// TIA Portal project "lab3" (V15)

(* hardware
DEVICE "S71500/ET200MP station_1"  S7-1500 station
   slot 0: "Rail_0"  Rack  6ES7 590-1***0-0AA0
   slot 1: "PLC_1"  CPU 1512C-1 PN  6ES7 512-1CK01-0AB0  V2.5
      slot 3: "CPU display_1"  6ES7591-1AA00-0AA0
*)

// ===== PLC "PLC_1"  CPU 1512C-1 PN =====

VAR_GLOBAL   // PLC tag table "Default tag table"
   "DIGITALNI_ULAZ_KLIP_1_LEVO_NC" AT %I10.0 : Bool;
   "DIGITALNI_ULAZ_KLIP_1_DESNO_NC" AT %I10.1 : Bool;
   "DIGITALNI_ULAZ_KLIP_2_LEVO_NO" AT %I10.2 : Bool;
   "DIGITALNI_ULAZ_KLIP_2_DESNO_NC" AT %I10.3 : Bool;
   "DIGITALNI_ULAZ_KLIP_3_LEVO_NO" AT %I10.4 : Bool;
   "DIGITALNI_ULAZ_KLIP_3_DESNO_NO" AT %I10.5 : Bool;
   "DIGITALNI_ULAZ_KLIP_4_LEVO_NC" AT %I10.6 : Bool;
   "DIGITALNI_ULAZ_KLIP_4_DESNO_NO" AT %I10.7 : Bool;
   "DIGITALNI_IZLAZ_KLIP_1_LEVO" AT %Q4.0 : Bool;
   "DIGITALNI_IZLAZ_KLIP_1_DESNO" AT %Q4.1 : Bool;
   "DIGITALNI_IZLAZ_KLIP_2_LEVO" AT %Q4.2 : Bool;
   "DIGITALNI_IZLAZ_KLIP_2_DESNO" AT %Q4.3 : Bool;
   "DIGITALNI_IZLAZ_KLIP_3_LEVO" AT %Q4.4 : Bool;
   "DIGITALNI_IZLAZ_KLIP_4_LEVO" AT %Q4.6 : Bool;
   "ANALOGNI_ULAZ_POZICIJA_KLIP_1" AT %IW0 : Word;
   "ANALOGNI_ULAZ_POZICIJA_KLIP_4" AT %IW2 : Word;
   "TIMER" AT %T0 : Timer;
   "COUNTER_INNER_LOOP" AT %C0 : Counter;
   "COUNTER_OUTER_LOOP" AT %C1 : Counter;
   "BROJAC_ODRZAVANJE_KLIP_4" AT %C2 : Counter;
END_VAR

DATA_BLOCK "DB"   // DB1
{ S7_Optimized_Access := 'TRUE' }
VERSION : 0.1
   VAR
      "POZICIJA_KLIP_30%" : Word := 8310;
      "POZICIJA_KLIP_40%" : Word := 11080;
      "POZICIJA_KLIP_50%" : Word := 13850;
      "POZICIJA_KLIP_70%" : Word := 19390;
      "POZICIJA_KLIP_90%" : Word := 24930;
      "POZICIJA_KLIP_80%" : Word := 22160;
      POZICIJA_MAX : Word := 27700;
   END_VAR
BEGIN
END_DATA_BLOCK

DATA_BLOCK "SEKVENCA_DB"   // DB2
{ S7_Optimized_Access := 'TRUE' }
VERSION : 0.1
// stored: InstanceOfName SEKVENCA
"SEKVENCA"
BEGIN
END_DATA_BLOCK

FUNCTION_BLOCK "SEKVENCA"   // FB1, GRAPH_PLUS
{ S7_Optimized_Access := 'TRUE' }
VERSION : 0.1
   VAR_INPUT
      OFF_SQ : Bool := false;   // Turn sequence off
      INIT_SQ : Bool := false;   // Set sequence to initial state
      ACK_EF : Bool := false;   // Acknowledge all errors and faults
      S_PREV : Bool := false;   // Output previous step in parameter S_NO
      S_NEXT : Bool := false;   // Indicate next step in parameter S_NO
      SW_AUTO : Bool := false;   // Automatic mode
      SW_TAP : Bool := false;   // Semiautomatic/switch with transition
      SW_TOP : Bool := false;   // Semiautomatic/ignore transition
      SW_MAN : Bool := false;   // Manual mode
      S_SEL : Int := 0;   // Select step to be output to S_NO
      S_ON : Bool := false;   // Activate step indicated in S_NO
      S_OFF : Bool := false;   // Deactivate step indicated S_NO
      T_PUSH : Bool := false;   // Enable transition to switch in semi automatic mode
   END_VAR
   VAR_OUTPUT
      S_NO : Int := 0;   // Step number
      S_MORE : Bool := false;   // More steps are available and can be shown in S_NO
      S_ACTIVE : Bool := false;   // Step indicated in S_NO is active
      ERR_FLT : Bool := false;   // Interlock or supervision group error
      AUTO_ON : Bool := false;   // Automatic mode is active
      TAP_ON : Bool := false;   // Semiautomatic mode/step with transition enabled
      TOP_ON : Bool := false;   // Semiautomatic mode/ignore transition enabled
      MAN_ON : Bool := false;   // Manual mode is active
   END_VAR
   VAR
      HMI_INFO : Array[0..14] of UInt;
      IF_PAR : G7_IfParPlus_V5;
      RT_DATA : G7_RTDataPlus_V5;   // Internal data area
      Trans1 : G7_TransitionPlus_V5;   // Transition structure
      Trans2 : G7_TransitionPlus_V5;   // Transition structure
      Trans3 : G7_TransitionPlus_V5;   // Transition structure
      Trans4 : G7_TransitionPlus_V5;   // Transition structure
      Trans5 : G7_TransitionPlus_V5;   // Transition structure
      Trans6 : G7_TransitionPlus_V5;   // Transition structure
      Trans7 : G7_TransitionPlus_V5;   // Transition structure
      Trans8 : G7_TransitionPlus_V5;   // Transition structure
      Trans9 : G7_TransitionPlus_V5;   // Transition structure
      Trans10 : G7_TransitionPlus_V5;   // Transition structure
      Trans11 : G7_TransitionPlus_V5;   // Transition structure
      Trans12 : G7_TransitionPlus_V5;   // Transition structure
      Trans13 : G7_TransitionPlus_V5;   // Transition structure
      INICIJALIZACIJA : G7_StepPlus_V5;   // Step structure
      Step1 : G7_StepPlus_V5;   // Step structure
      Step2 : G7_StepPlus_V5;   // Step structure
      ODRZAVANJE_KLIP_4_LEVO : G7_StepPlus_V5;   // Step structure
      ODRZAVANJE_KLIP_4_DESNO : G7_StepPlus_V5;   // Step structure
      Step3 : G7_StepPlus_V5;   // Step structure
      Step4 : G7_StepPlus_V5;   // Step structure
      Step5 : G7_StepPlus_V5;   // Step structure
      ODRZAVANJE_KLIP_1_DESNO : G7_StepPlus_V5;   // Step structure
      ODRZAVANJE_KLIP_1_LEVO : G7_StepPlus_V5;   // Step structure
      Step6 : G7_StepPlus_V5;   // Step structure
      Step7 : G7_StepPlus_V5;   // Step structure
      Step8 : G7_StepPlus_V5;   // Step structure
      Step9 : G7_StepPlus_V5;   // Step structure
      Step10 : G7_StepPlus_V5;   // Step structure
      SINI : Array[0..7] of USInt;
      LSTT : Array[0..12] of USInt;
      ATAJ : Array[0..12] of USInt;
      ATAB : Array[0..12] of USInt;
      PSTT : Array[0..12] of USInt;
      NSTT : Array[0..12] of USInt;
      ASSJ : Array[0..14] of USInt;
      ASSB : Array[0..14] of USInt;
      PTTS : Array[0..14] of USInt;
      NTTS : Array[0..14] of USInt;
      SW_SQTS : Array[0..14] of USInt;
      SWITCH : Array[0..7] of USInt;
      TVX : Array[0..11] of USInt;
      TTX : Array[0..11] of USInt;
      TSX : Array[0..7] of USInt;
      S00X : Array[0..7] of USInt;
      SOFFX : Array[0..7] of USInt;
      SONX : Array[0..7] of USInt;
      SAX : Array[0..7] of USInt;
      SERRX : Array[0..15] of USInt;
      SMX : Array[0..15] of USInt;
      S0X : Array[0..15] of USInt;
      S1X : Array[0..15] of USInt;
      IL_ALARM_INST : Diag_Alarm;
      SUP_ALARM_INST : Diag_Alarm;
      STEP_TIME_ALARM_INST : Diag_Alarm;
      IEC_TIMER_INST : IEC_TIMER;
      TRANSACTION_FLAG : Bool := false;
   END_VAR
   // SINI[0] := 2;
   // SINI[2] := 255;
   // SINI[3] := 255;
   // SINI[4] := 255;
   // LSTT[0] := 255;
   // LSTT[1] := 255;
   // LSTT[2] := 255;
   // LSTT[3] := 255;
   // LSTT[4] := 5;
   // LSTT[5] := 255;
   // ATAJ[1] := 1;
   // ATAJ[2] := 2;
   // ATAJ[3] := 3;
   // ATAJ[4] := 4;
   // ATAJ[5] := 5;
   // ATAB[1] := 1;
   // ATAB[2] := 2;
   // ATAB[3] := 3;
   // ATAB[4] := 5;
   // ATAB[5] := 4;
   // PSTT[1] := 1;
   // PSTT[2] := 2;
   // PSTT[3] := 5;
   // PSTT[4] := 6;
   // PSTT[5] := 6;
   // NSTT[0] := 1;
   // NSTT[1] := 2;
   // NSTT[2] := 5;
   // NSTT[3] := 6;
   // NSTT[4] := 5;
   // NSTT[5] := 7;
   // ASSJ[1] := 1;
   // ASSJ[2] := 2;
   // ASSJ[3] := 4;
   // ASSJ[4] := 13;
   // ASSJ[5] := 5;
   // ASSJ[6] := 6;
   // ASSB[1] := 1;
   // ASSB[2] := 3;
   // ASSB[3] := 4;
   // ASSB[4] := 2;
   // ASSB[5] := 5;
   // ASSB[6] := 6;
   // PTTS[0] := 255;
   // PTTS[2] := 1;
   // PTTS[3] := 1;
   // PTTS[4] := 1;
   // PTTS[5] := 2;
   // PTTS[6] := 3;
   // NTTS[1] := 1;
   // NTTS[2] := 2;
   // NTTS[3] := 10;
   // NTTS[4] := 10;
   // NTTS[5] := 3;
   // NTTS[6] := 5;
   // SW_SQTS[2] := 1;
   // SW_SQTS[3] := 2;
   // SW_SQTS[4] := 3;
   // SW_SQTS[5] := 1;
   // SW_SQTS[6] := 1;
   // SWITCH[2] := 122;
   // SWITCH[1] := 12;
   // TVX[0] := 16#1;
   // TTX[0] := 16#1;
   // TSX[0] := 16#1;
   // S00X[0] := 16#1;
   // SOFFX[0] := 16#1;
   // SONX[0] := 16#1;
   // SAX[0] := 16#1;
   // SERRX[0] := 16#1;
   // SMX[0] := 16#1;
   // S0X[0] := 16#1;
   // S1X[0] := 16#1;
   // SINI[5] := 255;
   // SINI[6] := 255;
   // SINI[7] := 255;
   // LSTT[6] := 255;
   // ATAJ[6] := 6;
   // ATAB[6] := 6;
   // PSTT[6] := 7;
   // NSTT[6] := 10;
   // ASSJ[7] := 7;
   // ASSJ[8] := 3;
   // ASSJ[9] := 8;
   // ASSB[7] := 9;
   // ASSB[8] := 7;
   // ASSB[9] := 8;
   // PTTS[7] := 5;
   // PTTS[8] := 5;
   // PTTS[9] := 5;
   // NTTS[7] := 6;
   // NTTS[8] := 10;
   // NTTS[9] := 10;
   // SW_SQTS[7] := 4;
   // SW_SQTS[8] := 5;
   // SW_SQTS[9] := 6;
   // SWITCH[3] := 118;
   // SWITCH[4] := 108;
   // SWITCH[5] := 92;
   // LSTT[7] := 255;
   // ATAJ[7] := 7;
   // ATAB[7] := 7;
   // PSTT[7] := 10;
   // NSTT[7] := 11;
   // ASSJ[10] := 10;
   // ASSB[10] := 10;
   // PTTS[10] := 6;
   // NTTS[10] := 7;
   // SW_SQTS[10] := 4;
   // LSTT[8] := 255;
   // LSTT[9] := 255;
   // LSTT[10] := 255;
   // LSTT[11] := 255;
   // LSTT[12] := 1;
   // ATAJ[8] := 8;
   // ATAJ[9] := 9;
   // ATAJ[10] := 10;
   // ATAJ[11] := 11;
   // ATAJ[12] := 12;
   // ATAB[8] := 8;
   // ATAB[9] := 9;
   // ATAB[10] := 10;
   // ATAB[11] := 12;
   // ATAB[12] := 11;
   // PSTT[8] := 12;
   // PSTT[9] := 11;
   // PSTT[10] := 13;
   // PSTT[11] := 14;
   // PSTT[12] := 14;
   // NSTT[8] := 13;
   // NSTT[9] := 12;
   // NSTT[10] := 14;
   // NSTT[11] := 255;
   // NSTT[12] := 1;
   // ASSJ[11] := 11;
   // ASSJ[12] := 12;
   // ASSJ[13] := 9;
   // ASSJ[14] := 14;
   // ASSB[11] := 11;
   // ASSB[12] := 12;
   // ASSB[13] := 13;
   // ASSB[14] := 14;
   // PTTS[11] := 7;
   // PTTS[12] := 9;
   // PTTS[13] := 8;
   // PTTS[14] := 10;
   // NTTS[11] := 9;
   // NTTS[12] := 8;
   // NTTS[13] := 10;
   // NTTS[14] := 11;
   // SW_SQTS[11] := 4;
   // SW_SQTS[12] := 4;
   // SW_SQTS[13] := 4;
   // SW_SQTS[14] := 7;
   // SWITCH[6] := 60;
BEGIN
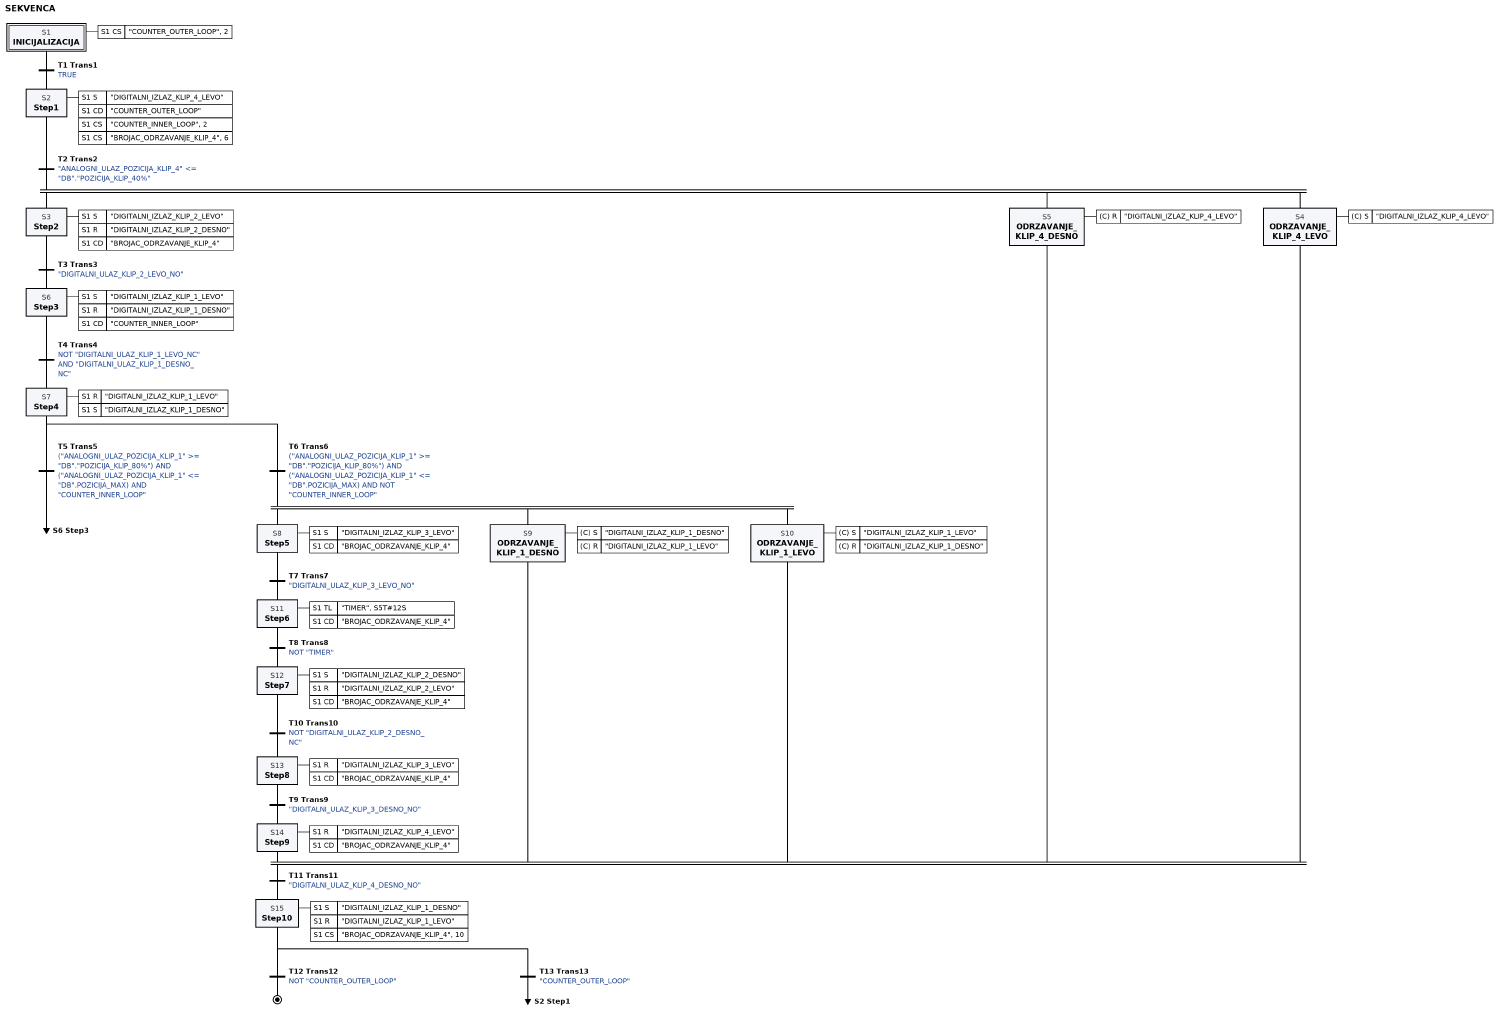
   // sequencer 1
   INITIAL_STEP INICIJALIZACIJA:   // S1, max time T#10S, warning time T#7S
          S1  CS   "COUNTER_OUTER_LOOP", 2
   END_STEP
   TRANSITION Trans1 FROM INICIJALIZACIJA TO Step1   // T1
      := TRUE;
   END_TRANSITION
   STEP Step2:   // S3, max time T#10S, warning time T#7S
          S1  S    "DIGITALNI_IZLAZ_KLIP_2_LEVO"
          S1  R    "DIGITALNI_IZLAZ_KLIP_2_DESNO"
          S1  CD   "BROJAC_ODRZAVANJE_KLIP_4"
   END_STEP
   TRANSITION Trans3 FROM Step2 TO Step3   // T3
      := "DIGITALNI_ULAZ_KLIP_2_LEVO_NO";
   END_TRANSITION
   STEP ODRZAVANJE_KLIP_4_DESNO:   // S5, max time T#10S, warning time T#7S
      interlock C := "ANALOGNI_ULAZ_POZICIJA_KLIP_4" <= "DB"."POZICIJA_KLIP_30%";
      (C)     R    "DIGITALNI_IZLAZ_KLIP_4_LEVO"
   END_STEP
   STEP ODRZAVANJE_KLIP_4_LEVO:   // S4, max time T#10S, warning time T#7S
      interlock C := ("ANALOGNI_ULAZ_POZICIJA_KLIP_4" >= "DB"."POZICIJA_KLIP_50%") AND ("ANALOGNI_ULAZ_POZICIJA_KLIP_4" <= "DB".POZICIJA_MAX) AND "BROJAC_ODRZAVANJE_KLIP_4";
      (C)     S    "DIGITALNI_IZLAZ_KLIP_4_LEVO"
   END_STEP
   STEP Step1:   // S2, max time T#10S, warning time T#7S
          S1  S    "DIGITALNI_IZLAZ_KLIP_4_LEVO"
          S1  CD   "COUNTER_OUTER_LOOP"
          S1  CS   "COUNTER_INNER_LOOP", 2
          S1  CS   "BROJAC_ODRZAVANJE_KLIP_4", 6
   END_STEP
   TRANSITION Trans2 FROM Step1 TO (Step2, ODRZAVANJE_KLIP_4_DESNO, ODRZAVANJE_KLIP_4_LEVO)   // T2
      := "ANALOGNI_ULAZ_POZICIJA_KLIP_4" <= "DB"."POZICIJA_KLIP_40%";
   END_TRANSITION
   STEP Step3:   // S6, max time T#10S, warning time T#7S
          S1  S    "DIGITALNI_IZLAZ_KLIP_1_LEVO"
          S1  R    "DIGITALNI_IZLAZ_KLIP_1_DESNO"
          S1  CD   "COUNTER_INNER_LOOP"
   END_STEP
   TRANSITION Trans4 FROM Step3 TO Step4   // T4
      := NOT "DIGITALNI_ULAZ_KLIP_1_LEVO_NC" AND "DIGITALNI_ULAZ_KLIP_1_DESNO_NC";
   END_TRANSITION
   STEP Step4:   // S7, max time T#10S, warning time T#7S
          S1  R    "DIGITALNI_IZLAZ_KLIP_1_LEVO"
          S1  S    "DIGITALNI_IZLAZ_KLIP_1_DESNO"
   END_STEP
   TRANSITION Trans5 FROM Step4 TO Step3   // T5, jump
      := ("ANALOGNI_ULAZ_POZICIJA_KLIP_1" >= "DB"."POZICIJA_KLIP_80%") AND ("ANALOGNI_ULAZ_POZICIJA_KLIP_1" <= "DB".POZICIJA_MAX) AND "COUNTER_INNER_LOOP";
   END_TRANSITION
   TRANSITION Trans6 FROM Step4 TO (Step5, ODRZAVANJE_KLIP_1_DESNO, ODRZAVANJE_KLIP_1_LEVO)   // T6
      := ("ANALOGNI_ULAZ_POZICIJA_KLIP_1" >= "DB"."POZICIJA_KLIP_80%") AND ("ANALOGNI_ULAZ_POZICIJA_KLIP_1" <= "DB".POZICIJA_MAX) AND NOT "COUNTER_INNER_LOOP";
   END_TRANSITION
   STEP Step5:   // S8, max time T#10S, warning time T#7S
          S1  S    "DIGITALNI_IZLAZ_KLIP_3_LEVO"
          S1  CD   "BROJAC_ODRZAVANJE_KLIP_4"
   END_STEP
   TRANSITION Trans7 FROM Step5 TO Step6   // T7
      := "DIGITALNI_ULAZ_KLIP_3_LEVO_NO";
   END_TRANSITION
   STEP ODRZAVANJE_KLIP_1_DESNO:   // S9, max time T#10S, warning time T#7S
      interlock C := "ANALOGNI_ULAZ_POZICIJA_KLIP_1" <= "DB"."POZICIJA_KLIP_70%";
      (C)     S    "DIGITALNI_IZLAZ_KLIP_1_DESNO"
      (C)     R    "DIGITALNI_IZLAZ_KLIP_1_LEVO"
   END_STEP
   TRANSITION Trans11 FROM (ODRZAVANJE_KLIP_4_DESNO, ODRZAVANJE_KLIP_4_LEVO, Step9, ODRZAVANJE_KLIP_1_LEVO, ODRZAVANJE_KLIP_1_DESNO) TO Step10   // T11
      := "DIGITALNI_ULAZ_KLIP_4_DESNO_NO";
   END_TRANSITION
   STEP ODRZAVANJE_KLIP_1_LEVO:   // S10, max time T#10S, warning time T#7S
      interlock C := ("ANALOGNI_ULAZ_POZICIJA_KLIP_1" >= "DB"."POZICIJA_KLIP_90%") AND ("ANALOGNI_ULAZ_POZICIJA_KLIP_1" <= "DB".POZICIJA_MAX);
      (C)     S    "DIGITALNI_IZLAZ_KLIP_1_LEVO"
      (C)     R    "DIGITALNI_IZLAZ_KLIP_1_DESNO"
   END_STEP
   STEP Step6:   // S11, max time T#10S, warning time T#7S
          S1  TL   "TIMER", S5T#12S
          S1  CD   "BROJAC_ODRZAVANJE_KLIP_4"
   END_STEP
   TRANSITION Trans8 FROM Step6 TO Step7   // T8
      := NOT "TIMER";
   END_TRANSITION
   STEP Step7:   // S12, max time T#10S, warning time T#7S
          S1  S    "DIGITALNI_IZLAZ_KLIP_2_DESNO"
          S1  R    "DIGITALNI_IZLAZ_KLIP_2_LEVO"
          S1  CD   "BROJAC_ODRZAVANJE_KLIP_4"
   END_STEP
   TRANSITION Trans10 FROM Step7 TO Step8   // T10
      := NOT "DIGITALNI_ULAZ_KLIP_2_DESNO_NC";
   END_TRANSITION
   STEP Step8:   // S13, max time T#10S, warning time T#7S
          S1  R    "DIGITALNI_IZLAZ_KLIP_3_LEVO"
          S1  CD   "BROJAC_ODRZAVANJE_KLIP_4"
   END_STEP
   TRANSITION Trans9 FROM Step8 TO Step9   // T9
      := "DIGITALNI_ULAZ_KLIP_3_DESNO_NO";
   END_TRANSITION
   STEP Step9:   // S14, max time T#10S, warning time T#7S
          S1  R    "DIGITALNI_IZLAZ_KLIP_4_LEVO"
          S1  CD   "BROJAC_ODRZAVANJE_KLIP_4"
   END_STEP
   STEP Step10:   // S15, max time T#10S, warning time T#7S
          S1  S    "DIGITALNI_IZLAZ_KLIP_1_DESNO"
          S1  R    "DIGITALNI_IZLAZ_KLIP_1_LEVO"
          S1  CS   "BROJAC_ODRZAVANJE_KLIP_4", 10
   END_STEP
   TRANSITION Trans12 FROM Step10 TO END   // T12
      := NOT "COUNTER_OUTER_LOOP";
   END_TRANSITION
   TRANSITION Trans13 FROM Step10 TO Step1   // T13, jump
      := "COUNTER_OUTER_LOOP";
   END_TRANSITION
END_FUNCTION_BLOCK

ORGANIZATION_BLOCK "Main"   // OB1, LAD, ProgramCycle
TITLE = "Main Program Sweep (Cycle)"
{ S7_Optimized_Access := 'TRUE' }
VERSION : 0.1
   VAR_INPUT
      Initial_Call : Bool;   // Initial call of this OB
      Remanence : Bool;   // =True, if remanent data are available
   END_VAR
BEGIN

REGION Network 1
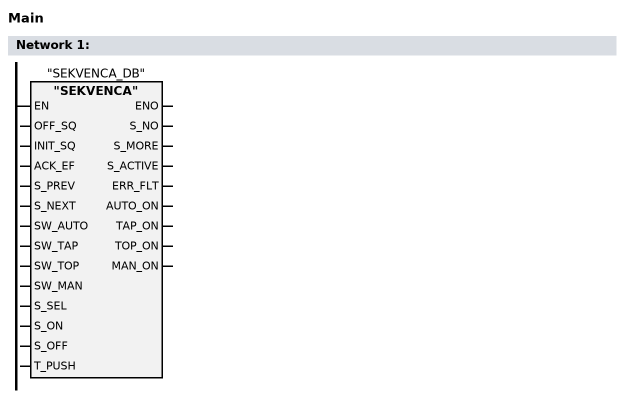
   RUNG wire#powerrail
      "SEKVENCA_DB"(OFF_SQ :=, INIT_SQ :=, ACK_EF :=, S_PREV :=, S_NEXT :=, SW_AUTO :=, SW_TAP :=, SW_TOP :=, SW_MAN :=, S_SEL :=, S_ON :=, S_OFF :=, T_PUSH :=, S_NO =>, S_MORE =>, S_ACTIVE =>, ERR_FLT =>, AUTO_ON =>, TAP_ON =>, TOP_ON =>, MAN_ON =>)
   END_RUNG
   // the same network as SCL:
   "SEKVENCA_DB"();   // "SEKVENCA"
END_REGION
END_ORGANIZATION_BLOCK